# EPICS substitutions: db/Beckhoff_3XXX/ecmcEL3174_+-10V.substitutions
file "ecmcEcSlave.template"
{
  pattern {}
          {}
}

#Actually the scalinging is between +-10.737V (see manual)
file "ecmcEX3XXX-chX.template"
{
  pattern {CH_ID, LINR,    ESLO,             EOFF,   EGU,        PREC, LOW,  LOLO,     HIGH,  HIHI,    HYST, LLSV,      LSV,     HSV,     HHSV   }
          {1,     "SLOPE", 3.2767723624E-4,  0,      "V",        3,    -10,  -10.5,    10,    10.5,    0,    "MAJOR",   "MINOR", "MINOR", "MAJOR"}
          {2,     "SLOPE", 3.2767723624E-4,  0,      "V",        3,    -10,  -10.5,    10,    10.5,    0,    "MAJOR",   "MINOR", "MINOR", "MAJOR"}
          {3,     "SLOPE", 3.2767723624E-4,  0,      "V",        3,    -10,  -10.5,    10,    10.5,    0,    "MAJOR",   "MINOR", "MINOR", "MAJOR"}
          {4,     "SLOPE", 3.2767723624E-4,  0,      "V",        3,    -10,  -10.5,    10,    10.5,    0,    "MAJOR",   "MINOR", "MINOR", "MAJOR"}
}
